FUNCTION_BLOCK DIV_DINT (* IEC 61131-3 DINT Division *)
  (* Standard: 61131-3 *)
  (* Version 0.0, 2004-12-15, JHC, Rockwell Automation, Converted from SRC format. *)
  (* Compiler header: package fb.rt.plc.math; *)
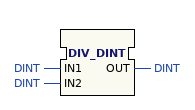
  VAR_INPUT
    IN1 : DINT; (* Dividend *)
    IN2 : DINT; (* Divisor *)
  END_VAR
  VAR_OUTPUT
    OUT : DINT; (* Quotient *)
  END_VAR
END_FUNCTION_BLOCK
